// TIA Portal project "第一次一条传送带" (V15.1)
// Vorlageprojekt für das Buch mit Zielsystem S7-1200

(* hardware
DEVICE "S7-1200-Station_1"  S7-1200 Station
   slot 0: "Baugruppenträger_0"  Rack  V1.0
   slot 1: "PLC_1"  CPU 1211C DC/DC/DC  6ES7 211-1AE40-0XB0  V4.1
*)

// ===== PLC "PLC_1"  CPU 1211C DC/DC/DC =====

VAR_GLOBAL   // PLC tag table "IO"
   "启动" AT %I0.0 : Bool;
   "暂停" AT %I0.1 : Bool;
   "停止" AT %I0.2 : Bool;
   "传感器" AT %I0.3 : Bool;
   "FACTORY I/O (Running)" AT %I0.4 : Bool;
   "绿灯" AT %Q0.0 : Bool;
   "黄灯" AT %Q0.1 : Bool;
   "红灯" AT %Q0.2 : Bool;
   "绿灯1" AT %Q0.3 : Bool;
   "黄灯1" AT %Q0.4 : Bool;
   "红灯1" AT %Q0.5 : Bool;
   "电机" AT %Q0.6 : Bool;
END_VAR

VAR_GLOBAL   // PLC tag table "中间标志位"
   "电机启动" AT %M0.0 : Bool;
END_VAR

FUNCTION "MHJ-PLC-Lab-Function-S71200" : Void   // FC9000, SCL
{ S7_Optimized_Access := 'TRUE' }
VERSION : 0.1
   VAR_TEMP
      rdTimeReturn : Int;
      outputTime : DTL;
      SyncVal : Byte;
      forVal : Int;
      forVal_2 : Int;
      Value : Byte;
   END_VAR
   VAR CONSTANT
      CompVal : Byte := 16#34;
      Value_01 : Byte := 16#11;
      Value_01_DW : DWord := 16#A165_D992;
      Value_02_DW : DWord := 16#58BE_4401;
   END_VAR
BEGIN

   #Value:=PEEK(area := 16#82,
        dbNumber := 0,
        byteOffset := 511);
   #Value := #Value + 1;

   POKE(area := 16#82,
        dbNumber := 0,
        byteOffset := 511,
        value := #Value);

   POKE(area:=16#81,
        dbNumber:=0,
        byteOffset:=1016,
        value:=#Value_01_DW);
   POKE(area := 16#81,
        dbNumber := 0,
        byteOffset := 1020,
        value := #Value_02_DW);

   POKE(area := 16#81,
        dbNumber := 0,
        byteOffset := 511,
        value := B#16#00);

   FOR #forVal := 0 TO 120 DO
       FOR #forVal_2:=0 TO 10 DO
           #rdTimeReturn:=RD_SYS_T(#outputTime);
           #rdTimeReturn := WR_SYS_T(#outputTime);
           #rdTimeReturn := RD_SYS_T(#outputTime);
           #rdTimeReturn := WR_SYS_T(#outputTime);
       END_FOR;
       #SyncVal:= PEEK(area := 16#81,
                      dbNumber := 0,
                      byteOffset := 511);
       IF #SyncVal = #CompVal THEN
          GOTO M_1;
       END_IF;
   END_FOR;
   RETURN;

   M_1:
   POKE(area := 16#81,
        dbNumber := 0,
        byteOffset := 511,
        value := B#16#0);
END_FUNCTION

ORGANIZATION_BLOCK "Main"   // OB1, LAD, ProgramCycle
TITLE = "Main Program Sweep (Cycle)"
{ S7_Optimized_Access := 'TRUE' }
VERSION : 0.1
   VAR_INPUT
      Initial_Call : Bool;   // Initial call of this OB
      Remanence : Bool;   // =True, if remanent data are available
   END_VAR
BEGIN

REGION Network 1: Konnektierungsbaustein für PLC-Lab
   // Im Netzwerk 1 wird der Konnektierungsbaustein für PLC-Lab aufgerufen.
   // Dieser Aufruf darf nicht entfernt werden!
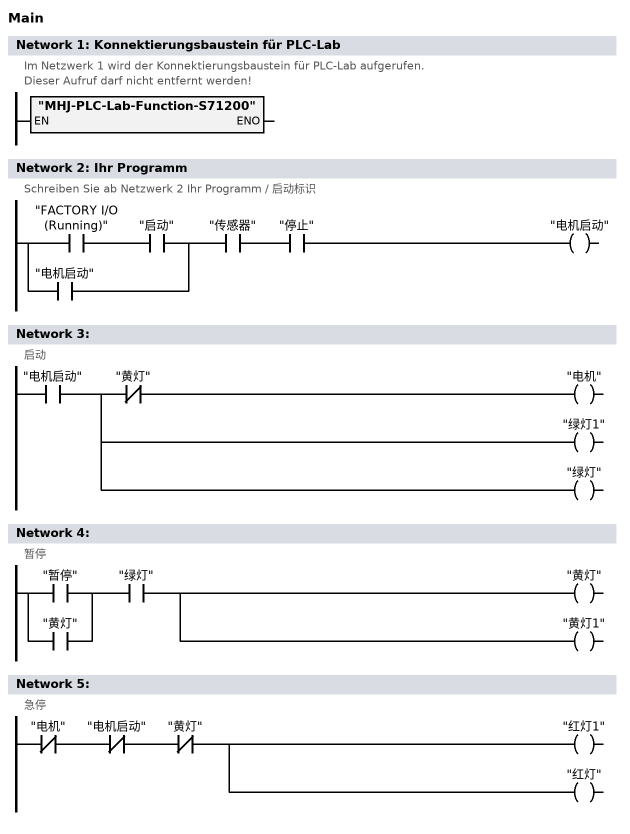
   RUNG wire#powerrail
      "MHJ-PLC-Lab-Function-S71200"()
   END_RUNG
   // the same network as SCL:
   "MHJ-PLC-Lab-Function-S71200"();
END_REGION

REGION Network 2: Ihr Programm
   // Schreiben Sie ab Netzwerk 2 Ihr Programm / 启动标识
   RUNG wire#powerrail
      Contact( "FACTORY I/O (Running)" )
      Contact( "启动" )
      wire#w1
      Contact( "传感器" )
      Contact( "停止" )
      Coil( "电机启动" )
   END_RUNG
   RUNG wire#powerrail
      Contact( "电机启动" )
   END_RUNG wire#w1
   // the same network as SCL:
   "电机启动" := (("FACTORY I/O (Running)" AND "启动") OR "电机启动") AND "传感器" AND "停止";
END_REGION

REGION Network 3
   // 启动
   RUNG wire#powerrail
      Contact( "电机启动" )
      wire#w1
      I_Contact( "黄灯" )
      Coil( "电机" )
   END_RUNG
   RUNG wire#w1
      Coil( "绿灯1" )
   END_RUNG
   RUNG wire#w1
      Coil( "绿灯" )
   END_RUNG
   // the same network as SCL:
   "电机" := "电机启动" AND NOT "黄灯";
   "绿灯1" := "电机启动";
   "绿灯" := "电机启动";
END_REGION

REGION Network 4
   // 暂停
   RUNG wire#powerrail
      Contact( "暂停" )
      wire#w1
      Contact( "绿灯" )
      wire#w2
      Coil( "黄灯" )
   END_RUNG
   RUNG wire#powerrail
      Contact( "黄灯" )
   END_RUNG wire#w1
   RUNG wire#w2
      Coil( "黄灯1" )
   END_RUNG
   // the same network as SCL:
   "黄灯" := ("暂停" OR "黄灯") AND "绿灯";
   "黄灯1" := "黄灯";
END_REGION

REGION Network 5
   // 急停
   RUNG wire#powerrail
      I_Contact( "电机" )
      I_Contact( "电机启动" )
      I_Contact( "黄灯" )
      wire#w1
      Coil( "红灯1" )
   END_RUNG
   RUNG wire#w1
      Coil( "红灯" )
   END_RUNG
   // the same network as SCL:
   "红灯1" := NOT "电机" AND NOT "电机启动" AND NOT "黄灯";
   "红灯" := "红灯1";
END_REGION
END_ORGANIZATION_BLOCK